Fanuc KAREL source: MSG_PING.kl

PROGRAM T
%NOLOCKGROUP
VAR
 v0 : STRING[40]
 v1 : INTEGER
BEGIN
 MSG_PING(v0, v1)
END T
